FUNCTION "SM_StateLastCall" : Bool
{ S7_Optimized_Access := 'FALSE' }
VERSION : 0.1
   VAR_IN_OUT
      inst : "typeSM";
   END_VAR


BEGIN
	#SM_StateLastCall := #inst.stateChanged AND (#inst.stateTime = 0);
END_FUNCTION

